// TIA Portal V17 export
// export: Created 2022-04-06T07:28:39.5415585Z, ExportSetting WithDefaults, DisplayName Totally Integrated Automation Portal, DisplayVersion V17, DisplayName TIA Portal Openness, DisplayVersion V17, DisplayName TIA Portal Version Control Interface, DisplayVersion V17, DisplayName TIA Portal Test Suite Advanced, DisplayVersion V17, DisplayName SINAMICS Startdrive Advanced, DisplayVersion V17, DisplayName SINAMICS Startdrive G130, G150, S120, S150, SINAMICS MV, S210, DisplayVersion V17, DisplayName SINAMICS Startdrive G110M, G120, G120C, G120D, G120P, G115D, DisplayVersion V17, DisplayName STEP 7 Professional, DisplayVersion V17, DisplayName STEP 7 Safety, DisplayVersion V17, DisplayName WinCC Advanced / Unified PC, DisplayVersion V17
DATA_BLOCK "SLI_gDB_FileHandling"   // DB11
{ S7_Optimized_Access := 'FALSE' }
VERSION : 0.1
// stored: AutoNumber true, DBAccessibleFromOPCUA true, DBAccessibleFromWebserver true, IsOnlyStoredInLoadMemory false, IsWriteProtectedInAS false
   VAR
      "name" : String := 'UserFiles/SLI_text.txt';
      fileWrite : "typeFileReadWrite";
      fileRead { S7_SetPoint := 'True'} : "typeFileReadWrite";
      fileDelete { S7_SetPoint := 'True'} : "typeFileReadWrite";
      data2 { S7_SetPoint := 'True'} : Array[0..999] of Byte;
   END_VAR
BEGIN
   fileWrite.length := 1000;
   fileWrite.data[0] := 16#10;
   fileWrite.data[1] := 11;
   fileWrite.data[2] := 12;
   fileWrite.data[3] := 13;
   fileWrite.data[4] := 14;
   fileWrite.data[5] := 15;
   fileWrite.data[6] := 16;
   fileWrite.data[7] := 17;
   fileWrite.data[8] := 18;
   fileWrite.data[9] := 19;
   fileWrite.data[10] := 20;
   data2[0] := 16#1;
   data2[1] := 2;
   data2[2] := 3;
   data2[3] := 4;
   data2[4] := 5;
   data2[5] := 6;
   data2[6] := 7;
   data2[7] := 8;
   data2[8] := 9;
   data2[9] := 10;
   data2[104] := 100;
END_DATA_BLOCK
